FUNCTION_BLOCK FB_PU_Zustandscheck
VAR_IN_OUT
	Zustand		: ST_PU_Zustand;
END_VAR
VAR_INPUT
	Steuerung		: ST_PU_Steuerung;
END_VAR
VAR_OUTPUT
END_VAR
VAR
	Timer1	: TON;
	Timer2	: TON;
	bWarnung1	: BOOL;
	bWarnung2	: BOOL;
END_VAR

(*
	Stoerung_Code
		0:	Allgemein Störung Pumpe (intern)
		1:	..
		2:	..
		3:
		4:
		5:
		6:
		7:

	Warnung_Code
		0:	Allgemein Warnung Pumpe (intern)
		1:	keine Betriebsrückmeldung
		2:	kein Volumenstrom
		3:	Pumpe im Handbetrieb
		4:
		5:
		6:
		7:

	Freigabe_Code
		0:	Freigabe durch Automatik entzogen
		1:	Freigabe durch Manuell entzogen
		2:	Freigabe durch Stoerung entzogen
*)
(* Interne Stoerungen / Warnungen *)

(* Warnung - keine Betriebsrückmeldung trotz Betriebsanforderung nach 1 Minute *)
IF (Zustand.Betrieb_Soll <> Zustand.Betrieb) THEN
	bWarnung1	:= TRUE;
ELSE
	bWarnung1	:= FALSE;
END_IF;
Timer1(	IN := bWarnung1,
		PT := T#1M,
		Q => Zustand.Warnung_Code.1
);

(* Warnung - kein Volumenstrom im Betrieb nach 1 Minute *)
IF (Zustand.Volumenstrom <= 0 AND Zustand.Betrieb) THEN
	bWarnung2	:= TRUE;
ELSE
	bWarnung2	:= FALSE;
END_IF;
Timer2(	IN := bWarnung2,
		PT := T#1M,
		Q => Zustand.Warnung_Code.2
);

(* Warnung - Pumpe im Handbetrieb *)
IF (Zustand.Modul_Betriebsart > 0) THEN
	Zustand.Warnung_Code.3	:= TRUE;
ELSE
	Zustand.Warnung_Code.3	:= FALSE;
END_IF;


(* ------------------------------------------------------------------- *)
(* Stoermeldung *)
IF Zustand.Stoerung_Code > 0 THEN
	Zustand.Stoerung := TRUE;
(*ELSE - wird nur durch Quittierung gelöscht
	Zustand.Stoerung := FALSE; *)
END_IF;

(* Warnmeldung *)
IF Zustand.Warnung_Code > 0 THEN
	Zustand.Warnung := TRUE;
ELSE
	Zustand.Warnung := FALSE;
END_IF;


(* ----- Freigabe_Code -------- *)
Zustand.Freigabe_Code.0 := NOT(Steuerung.Freigabe.auto);
Zustand.Freigabe_Code.1 := Steuerung.Freigabe.manu_Modus AND NOT Steuerung.Freigabe.manu;
Zustand.Freigabe_Code.2 := Zustand.Stoerung;

(* Freigabe *)
IF (Zustand.Freigabe_Code > 0 OR NOT Steuerung.Freigabe.auto ) THEN
	Steuerung.Freigabe.auto := FALSE;
ELSE
	Steuerung.Freigabe.auto := TRUE;
END_IF;

END_FUNCTION_BLOCK

(* stored: Version 1.1.0.1, ProductVersion 3.1.4024.9
   POU FB_PU_Zustandscheck: Id {ef154bd9-c0cd-4b28-8733-66caba65966f}, SpecialFunc None *)
